(* PLC project assembly_line, Bilinmeyen auto_fault 1, author 1337leets *)
(* stored: creationDateTime 2026-04-03T14:25:40, modificationDateTime 2026-04-06T11:02:48 *)

PROGRAM assembly
  VAR_INPUT
    SensorIn : BOOL;
    SensorMiddle : BOOL;
    SensorOut : BOOL;
    StartButton : BOOL;
    StopButton : BOOL;
    ResetButton : BOOL;
  END_VAR
  VAR_OUTPUT
    ConveyorMotor : BOOL;
    AlarmJam : BOOL;
  END_VAR
  VAR
    TONWait : TON;
    TONJam : TON;
    CTUIn : CTU;
    CTUOut : CTU;
    WaitDone : BOOL;
    Jammed : BOOL;
    ErrorState : BOOL;
    IODiff : INT;
    DiffAlarm : BOOL;
    AutoReset : BOOL;
    ResetState : BOOL;
  END_VAR
  VAR  (* added by the conversion: wires and edge detectors of the diagram *)
    R_TRIG1 : R_TRIG;
    R_TRIG2 : R_TRIG;
    R_TRIG3 : R_TRIG;
    R_TRIG4 : R_TRIG;
  END_VAR

(* LD diagram, written out as Structured Text *)
ConveyorMotor := (StartButton OR ConveyorMotor) AND NOT StopButton AND (SensorIn AND NOT SensorMiddle OR WaitDone) AND NOT ErrorState;
TONWait(IN := SensorMiddle, PT := T#2s);
WaitDone := TONWait.Q;
TONJam(IN := SensorMiddle, PT := T#5s);
Jammed := TONJam.Q;
R_TRIG1(CLK := SensorIn);
R_TRIG2(CLK := R_TRIG1.Q);
CTUIn(CU := R_TRIG2.Q, R := ResetState, PV := 5002);
R_TRIG3(CLK := SensorOut);
R_TRIG4(CLK := R_TRIG3.Q);
CTUOut(CU := R_TRIG4.Q, R := ResetState, PV := 5000);
IODiff := CTUIn.CV - CTUOut.CV;
DiffAlarm := IODiff >= 3;
ErrorState := (Jammed OR DiffAlarm OR ErrorState) AND NOT ResetButton;
AlarmJam := ErrorState;
ResetState := ResetButton OR AutoReset;
AutoReset := CTUOut.Q AND NOT DiffAlarm;
END_PROGRAM

CONFIGURATION Config0
  RESOURCE Res0 ON PLC
    TASK task0(INTERVAL := T#20ms, PRIORITY := 0);
    PROGRAM instance0 WITH task0 : assembly;
  END_RESOURCE
END_CONFIGURATION
